// TIA Portal V15.1 export
// export: Created 2024-05-17T05:38:36.1997139Z, ExportSetting WithDefaults, DisplayName Totally Integrated Automation Portal, DisplayVersion V15.1 Update 5, DisplayName TIA Portal Openness, DisplayVersion V15.1 Update 5, DisplayName SINAMICS Startdrive Advanced, DisplayVersion V15.1, DisplayName G130, G150, S120, S150, SINAMICS MV, S210, DisplayVersion V15.1, DisplayName G110M, G120, G120C, G120D, G120P, DisplayVersion V15.1, DisplayName STEP 7 Professional, DisplayVersion V15.1 Update 5, DisplayName STEP 7 Safety, DisplayVersion V15.1, DisplayName WinCC Professional, DisplayVersion V15.1 Update 5, DisplayName SIMATIC Visualization Architect, DisplayVersion V15.1
FUNCTION_BLOCK "LProcPAC-Conversion"   // FB1743, SCL
TITLE = LProcPAC-Conversion
{ S7_Optimized_Access := 'TRUE' }
AUTHOR : CSTAAL
VERSION : 2.0
// stored: AutoNumber false, IsIECCheckEnabled false, IsRetainMemResEnabled false, MemoryReserve 100, SetENOAutomatically False, UDAEnableTagReadback false
   VAR_INPUT
      id_hdword { ExternalAccessible := 'False'; ExternalVisible := 'False'; ExternalWritable := 'False'} : DWord := DWORD#16#0000_0000;   // highdword of the 64Bit number
      id_ldword { ExternalAccessible := 'False'; ExternalVisible := 'False'; ExternalWritable := 'False'} : DWord := DWORD#16#0000_0000;   // lowdword of the 64Bit number
   END_VAR
   VAR_OUTPUT
      FINE { ExternalAccessible := 'False'; ExternalVisible := 'False'; ExternalWritable := 'False'} : DInt := 0;   // counter value fine
      RAW { ExternalAccessible := 'False'; ExternalVisible := 'False'; ExternalWritable := 'False'} : DInt := 0;   // counter value raw
      ERROR { ExternalAccessible := 'False'; ExternalVisible := 'False'; ExternalWritable := 'False'} : Word := WORD#16#0000;   // error word of the function block
   END_VAR
   VAR DB_SPECIFIC
      sCounterval { ExternalAccessible := 'False'; ExternalVisible := 'False'; ExternalWritable := 'False'} : Struct   // 64Bit structure
         hdword { ExternalAccessible := 'False'; ExternalVisible := 'False'; ExternalWritable := 'False'} : DWord := DWORD#16#0000_0000;   // highdword of the 64Bit number
         ldword { ExternalAccessible := 'False'; ExternalVisible := 'False'; ExternalWritable := 'False'} : DWord := DWORD#16#0000_0000;   // lowdword of the 64Bit number
      END_STRUCT;
   END_VAR
   VAR
      vwords AT sCounterval : Struct   // AT sCounterval : STRUCT
         HDHW : Word;   // highword of the highdword of the 64Bit number
         HDLW : Word;   // lowword of the highdword of the 64Bit number
         LDHW : Word;   // highword of the lowdword of the 64Bit number
         LDLW : Word;   // lowword of the lowdword of the 64Bit number
      END_STRUCT;
      sVZ { ExternalAccessible := 'False'; ExternalVisible := 'False'; ExternalWritable := 'False'} : Word := WORD#16#0000;   // algebraic sign of the 64Bit number
      sCH { ExternalAccessible := 'False'; ExternalVisible := 'False'; ExternalWritable := 'False'} : Word := WORD#16#0000;   // exponent of the 64Bit number
      sExp { ExternalAccessible := 'False'; ExternalVisible := 'False'; ExternalWritable := 'False'} : Int := 0;   // exponent of the 64Bit number
      sResDiv { ExternalAccessible := 'False'; ExternalVisible := 'False'; ExternalWritable := 'False'} : DWord := DWORD#16#0000_0000;   // result of division
      sDivision { ExternalAccessible := 'False'; ExternalVisible := 'False'; ExternalWritable := 'False'} : DWord := DWORD#16#0000_0000;   // dword for division of 1.000.000.000
      sFINE { ExternalAccessible := 'False'; ExternalVisible := 'False'; ExternalWritable := 'False'} : DInt := 0;   // static counter falue fine
      sRAW { ExternalAccessible := 'False'; ExternalVisible := 'False'; ExternalWritable := 'False'} : DInt := 0;   // static counter value raw
      sERROR { ExternalAccessible := 'False'; ExternalVisible := 'False'; ExternalWritable := 'False'} : Word := WORD#16#0000;   // static error word
      i { ExternalAccessible := 'False'; ExternalVisible := 'False'; ExternalWritable := 'False'} : Int := 0;   // loop counter
   END_VAR
   VAR CONSTANT
      cBIAS : Word := WORD#16#03FF;   // 03FFh --> 1023dez ... bias of the 64Bit number
      cVZmask : Word := WORD#16#8000;   // mask to seperate the algebraic sign
      cCHmask : Word := WORD#16#7FF0;   // mask to seperate the exponent field
      cMTmask : DWord := DWORD#16#000F_FFFF;   // mask to seperate the mantissa
      cMask : DWord := DWORD#16#0000_0001;   // general mask
      cNrGIGA : DInt := 1_000_000_000;   // 1.000.000.000(dez)
      cNrKILO : Int := 1000;   // 1.000(dez)
   END_VAR
BEGIN



   (***********************************************************************************************
   ********************************************  CODE  *******************************************
   ***********************************************************************************************)

   // initialization of internal variables
   // allocation of the two dwords of the energy counter value
   #sCounterval.hdword := #id_hdword;
   #sCounterval.ldword := #id_ldword;
   #sResDiv := dw#16#000000000;

   // seperate VZ (sign bit)
   #sVZ := #vwords.HDHW AND #cVZmask;

   // seperate CH (exponent field with offset(cBias))
   // seperate exponent of the 64Bit value
   #sCH := SHR(IN := (#vwords.HDHW AND #cCHmask), N := 4);
   #sExp := WORD_TO_INT(#sCH) - WORD_TO_INT(#cBIAS);

   // check the algebraic sign
   // negative counter values indicate an error
   IF #sVZ = #cVZmask
   THEN
       #sERROR := w#16#0001;
   ELSE
       // check the special case of the 0 value and the value < 1
       // the output values have the format dint --> 0,1 is not possible
       IF #sCH = w#16#0000 OR WORD_TO_INT(#sCH) < WORD_TO_INT(#cBIAS)
       THEN
           #sFINE := 0;
           #sRAW := 0;
       ELSE
           // **************************
           // ********** FINE **********
           // **************************

           // *** If the exponent is smaller than 29 the number is smaller than 1.000.000.000
           // *** You have to seperate the valid bits (sExp)of the mantissa
           // *** At the end you have to add the hidden 1 Bit
           IF #sExp < 29
           THEN
               IF #sExp < 20
               THEN
                   #sFINE := DWORD_TO_DINT(SHR(IN := (#sCounterval.hdword AND #cMTmask), N := 20 - #sExp) OR SHL(IN := #cMask, N := #sExp));

               ELSIF #sExp = 20
               THEN
                   #sFINE := DWORD_TO_DINT(#sCounterval.hdword AND #cMTmask OR SHL(IN := #cMask, N := 20));
               ELSE
                   #sFINE := DWORD_TO_DINT((SHL(IN := (#sCounterval.hdword AND #cMTmask), N := #sExp - 20) OR SHR(IN := #sCounterval.ldword, N := 32 - (#sExp - 20))) OR SHL(IN := #cMask, N := #sExp));
               END_IF;

               // *** If the exponent is 29 the number is between 536.870.912 and 1.073.741.823
               // *** You have to subtract 1.000.000.000 if it's bigger than 1.000.000.000
               // *** The result ist the fine counter value
           ELSIF #sExp = 29
           THEN
               IF DWORD_TO_DINT((SHL(IN := (#sCounterval.hdword AND #cMTmask), N := #sExp - 20) OR SHR(IN := #sCounterval.ldword, N := 32 - (#sExp - 20))) OR SHL(IN := #cMask, N := #sExp)) > #cNrGIGA
               THEN
                   #sFINE := DWORD_TO_DINT((SHL(IN := (#sCounterval.hdword AND #cMTmask), N := #sExp - 20) OR SHR(IN := #sCounterval.ldword, N := 32 - (#sExp - 20))) OR SHL(IN := #cMask, N := #sExp)) - #cNrGIGA;

               ELSIF DWORD_TO_DINT((SHL(IN := (#sCounterval.hdword AND #cMTmask), N := #sExp - 20) OR SHR(IN := #sCounterval.ldword, N := 32 - (#sExp - 20))) OR SHL(IN := #cMask, N := #sExp)) = #cNrGIGA
               THEN
                   #sFINE := 0;
               ELSE
                   #sFINE := DWORD_TO_DINT((SHL(IN := (#sCounterval.hdword AND #cMTmask), N := #sExp - 20) OR SHR(IN := #sCounterval.ldword, N := 32 - (#sExp - 20))) OR SHL(IN := #cMask, N := #sExp));
               END_IF;

               // *** If the exponent is bigger then 29 you have to divide the number by 1.000.000.000
               // *** the rest of the division is the fine counter value
           ELSE
               #sDivision := (SHL(IN := (#sCounterval.hdword AND #cMTmask), N := 9) OR SHR(IN := #sCounterval.ldword, N := 23)) OR SHL(IN := #cMask, N := 29);
               FOR #i := 0 TO #sExp - 29 DO
                   IF DWORD_TO_DINT(#sDivision) > #cNrGIGA OR DWORD_TO_DINT(#sDivision) = #cNrGIGA
                   THEN

                       #sDivision := DINT_TO_DWORD(DWORD_TO_DINT(#sDivision) - #cNrGIGA);
                       IF #i <> #sExp - 29
                       THEN
                           #sDivision := SHL(IN := #sDivision, N := 1) OR (SHR(IN := #sCounterval.ldword, N := 22 - #i) AND #cMask);
                       ELSE
                           ;
                       END_IF;

                       #sResDiv := SHL(IN := #sResDiv, N := 1) OR dw#16#00000001;
                   ELSE
                       IF #i <> #sExp - 29
                       THEN
                           #sDivision := SHL(IN := #sDivision, N := 1) OR (SHR(IN := #sCounterval.ldword, N := 22 - #i) AND #cMask);
                       ELSE
                           ;
                       END_IF;

                       #sResDiv := SHL(IN := #sResDiv, N := 1);
                   END_IF;

               END_FOR;

               #sFINE := DWORD_TO_DINT(#sDivision);

           END_IF;

           // **************************
           // ********** RAW ***********
           // **************************

           // Initialisation of sResDiv for new division
           #sResDiv := dw#16#00000000;

           // *** If the exponent is smaller than 9 the number is smaller than 1.000
           // *** The raw counter value is 0
           IF #sExp < 9
           THEN
               #sRAW := 0;

               // *** If the exponent is 9 the number is between 512 and 1.023
               // *** You have to subtract 1.000
               // *** The result ist the raw counter value
           ELSIF #sExp = 9
           THEN
               IF DWORD_TO_DINT(SHR(IN := (#sCounterval.hdword AND #cMTmask), N := 20 - #sExp) OR SHL(IN := #cMask, N := #sExp)) > #cNrKILO
               THEN
                   #sRAW := 1;
               ELSE
                   #sRAW := 0;
               END_IF;

               // *** If the exponent is bigger then 29 you have to divide the number by 1.000.000.000
               // *** the result of the division is the raw countervalue
           ELSE
               #sDivision := SHR(IN := (#sCounterval.hdword AND #cMTmask), N := 11) OR SHL(IN := #cMask, N := 9);
               FOR #i := 0 TO #sExp - 9 DO
                   IF DWORD_TO_DINT(#sDivision) > #cNrKILO OR DWORD_TO_DINT(#sDivision) = #cNrKILO
                   THEN

                       #sDivision := DINT_TO_DWORD(DWORD_TO_DINT(#sDivision) - #cNrKILO);
                       IF #i <> #sExp - 9
                       THEN
                           #sDivision := SHL(IN := #sDivision, N := 1);
                           IF #i <= 10
                           THEN
                               #sDivision := #sDivision OR (SHR(IN := #sCounterval.hdword, N := 11 - (#i + 1)) AND #cMask);
                           ELSE
                               #sDivision := #sDivision OR (SHR(IN := #sCounterval.ldword, N := 32 - ((#i + 1) - 11)) AND #cMask);
                           END_IF;

                       ELSE
                           ;
                       END_IF;

                       #sResDiv := SHL(IN := #sResDiv, N := 1) OR dw#16#00000001;
                   ELSE
                       IF #i <> #sExp - 9
                       THEN
                           #sDivision := SHL(IN := #sDivision, N := 1);
                           IF #i <= 10
                           THEN
                               #sDivision := #sDivision OR (SHR(IN := #sCounterval.hdword, N := 11 - (#i + 1)) AND #cMask);
                           ELSE
                               #sDivision := #sDivision OR (SHR(IN := #sCounterval.ldword, N := 32 - ((#i + 1) - 11)) AND #cMask);
                           END_IF;

                       ELSE
                           ;
                       END_IF;

                       #sResDiv := SHL(IN := #sResDiv, N := 1);
                   END_IF;

               END_FOR;

               #sRAW := DWORD_TO_DINT(#sResDiv);

           END_IF;

       END_IF;
       #sERROR := w#16#0000;
   END_IF;

   #FINE := #sFINE;
   #RAW := #sRAW;
   #ERROR := #sERROR;
END_FUNCTION_BLOCK
